// TIA Portal V16 export
// export: Created 2024-04-10T09:00:39.579945Z, ExportSetting WithDefaults, DisplayName Totally Integrated Automation Portal, DisplayVersion V16 Update 6, DisplayName TIA Portal Version Control Interface, DisplayVersion V16 Update 2, DisplayName TIA Portal Openness, DisplayVersion V16 Update 6, DisplayName TIA Portal Test Suite Advanced, DisplayVersion V16, DisplayName SINAMICS Startdrive Advanced, DisplayVersion V16 Update 5, DisplayName SINAMICS Startdrive G130, G150, S120, S150, SINAMICS MV, S210, DisplayVersion V16 Update 5, DisplayName SINAMICS Startdrive G110M, G120, G120C, G120D, G120P, G115D, DisplayVersion V16 Update 5, DisplayName STEP 7 Professional, DisplayVersion V16 Update 6, DisplayName STEP 7 Safety, DisplayVersion V16, DisplayName WinCC Advanced, DisplayVersion V16 Update 6
FUNCTION_BLOCK "RH_OUT_1020MU"   // FB40, LAD
TITLE = Set receiver 865MU1020 outputs / Kuljetinpohja
{ S7_Optimized_Access := 'TRUE' }
AUTHOR : JLA
VERSION : 0.1
// stored: AutoNumber true, IsIECCheckEnabled false, IsRetainMemResEnabled false, MemoryReserve 100, SetENOAutomatically false, UDAEnableTagReadback false
   VAR
      Diag : "RMP_UDT_DIAG";   // Device diagnostics / Laitteen diagnostiikka
      Status : "RMP_UDT_DEV_STATUS";   // Device status information / Laitteen tilatieto
      HMI_Status : "RMP_HMI_DEV_STATUS";   // Device status information for HMI
      IO : Struct   // Device inputs and outputs / Laitteen tulot ja lähdöt
         Input : Struct
            Extended : Bool;   // Receiver extended / Kuljettimen turvakytkin
            Retracted : Bool;   // Receiver retracted / Tulovalokenno
            Rolls_coming : Bool;   // Rolls coming to receiver / Poistovalokenno
            Rolls_received : Bool;   // All rolls received / Rulla viivakoodin lukukohdassa
            Man_extend : Bool;   // Manual, receiver extend
            Man_retract : Bool;   // Manual, receiver retract / Seuraavan kuljettimen tulokenno
            Rolls_on_floor : Bool;   // Edellisen kuljettimen poistokenno / Rolls on floor before stopper
            Lidar_Field1 : Bool;   // Area between stop 1010 and Rm
            Lidar_Field2 : Bool;   // Area after stop 1010
            Lidar_Field3 : Bool;   // Conveyor 2030
            In_11 : Bool;
            In_12 : Bool;
            In_13 : Bool;
            In_14 : Bool;
            In_15 : Bool;
            In_16 : Bool;
            In_17 : Bool;
            In_18 : Bool;
            In_19 : Bool;
            In_20 : Bool;
            In_21 : Bool;
            In_22 : Bool;
            In_23 : Bool;
            In_24 : Bool;
            In_25 : Bool;
            In_26 : Bool;
            In_27 : Bool;
            In_28 : Bool;
            In_29 : Bool;
            In_30 : Bool;
            In_31 : Bool;
            In_32 : Bool;
         END_STRUCT;
         Output : Struct
            Receiver_extend : Bool;   // Receiver extend
            Receiver_retract : Bool;   // Receiver retract
            Out_3 : Bool;
            Out_4 : Bool;
            Out_5 : Bool;
            Out_6 : Bool;
            Out_7 : Bool;
            Out_8 : Bool;
            Out_9 : Bool;
            Out_10 : Bool;
            Out_11 : Bool;
            Out_12 : Bool;
            Out_13 : Bool;
            Out_14 : Bool;
            Out_15 : Bool;
            Out_16 : Bool;
            Out_17 : Bool;
            Out_18 : Bool;
            Out_19 : Bool;
            Out_20 : Bool;
            Out_21 : Bool;
            Out_22 : Bool;
            Out_23 : Bool;
            Out_24 : Bool;
            Out_25 : Bool;
            Out_26 : Bool;
            Out_27 : Bool;
            Out_28 : Bool;
            Out_29 : Bool;
            Out_30 : Bool;
            Out_31 : Bool;
            Out_32 : Bool;
         END_STRUCT;
      END_STRUCT;
      Flags : Struct   // Device auxilary flags / Laitteen apubitit
         Speed_1 : Bool;   // Speed selection 1 / Nopeusvalinta 1
         Speed_2 : Bool;   // Speed selection 2 / Nopeusvalinta 2
         Speed_3 : Bool;   // Speed selection 3 / Nopeusvalinta 3
         Speed_4 : Bool;   // Speed selection 4 / Nopeusvalinta 4
         Data_ok : Bool;   // Roll data present / Rulladata löytyy
         Entry_pec_fault : Bool;   // Entry pec fault bit
         Exit_pec_fault : Bool;   // Exit pec fault bit
         Auto_help : Bool;   // Auto status help bit
         Buffering : Bool;   // Buffering rolls on conveyor
         Separate : Bool;   // Separating rolls at conveyor exit joint
         Separate_p : Bool;   // Separating rolls at conveyor exit joint pulse
         Stopped : Bool;   // Device stopped
         Receiving : Bool;   // Receiving set on conveyor
         Bit_13 : Bool;
         Bit_14 : Bool;
         Bit_15 : Bool;
         Bit_16 : Bool;
         Bit_17 : Bool;
         Bit_18 : Bool;
         Bit_19 : Bool;
         Bit_20 : Bool;
         Bit_21 : Bool;
         Bit_22 : Bool;
         Bit_23 : Bool;
         Bit_24 : Bool;
         Bit_25 : Bool;
         Bit_26 : Bool;
         Bit_27 : Bool;
         Bit_28 : Bool;
         Bit_29 : Bool;
         Bit_30 : Bool;
         Bit_31 : Bool;
         Bit_32 : Bool;
         Bit_33 : Bool;
         Bit_34 : Bool;
         Bit_35 : Bool;
         Bit_36 : Bool;
         Bit_37 : Bool;
         Bit_38 : Bool;
         Bit_39 : Bool;
         Bit_40 : Bool;
         Bit_41 : Bool;
         Bit_42 : Bool;
         Bit_43 : Bool;
         Bit_44 : Bool;
         Bit_45 : Bool;
         Bit_46 : Bool;
         Bit_47 : Bool;
         Bit_48 : Bool;
         Bit_49 : Bool;
         Bit_50 : Bool;
         Bit_51 : Bool;
         Bit_52 : Bool;
         Bit_53 : Bool;
         Bit_54 : Bool;
         Bit_55 : Bool;
         Bit_56 : Bool;
         Bit_57 : Bool;
         Bit_58 : Bool;
         Bit_59 : Bool;
         Bit_60 : Bool;
         Bit_61 : Bool;
         Bit_62 : Bool;
         Bit_63 : Bool;
      END_STRUCT;
      Data : Struct   // Device data / Laitteen data
         Data_int_1 : Int;
         Data_int_2 : Int;
         Data_int_3 : Int;
         Data_int_4 : Int;
         Data_int_5 : Int;
         Data_int_6 : Int;
         Data_int_7 : Int;
         Data_int_8 : Int;
         Data_int_9 : Int;
         Data_int_10 : Int;
         Data_int_11 : Int;
         Data_int_12 : Int;
         Data_int_13 : Int;
         Data_int_14 : Int;
         Data_int_15 : Int;
         Data_int_16 : Int;
         Data_int_17 : Int;
         Data_int_18 : Int;
         Data_int_19 : Int;
         Data_int_20 : Int;
         Data_Dint_1 : DInt;
         Data_Dint_2 : DInt;
         Data_Dint_3 : DInt;
         Data_Dint_4 : DInt;
         Data_Dint_5 : DInt;
         Data_Dint_6 : DInt;
         Data_Dint_7 : DInt;
         Data_Dint_8 : DInt;
         Data_Dint_9 : DInt;
         Data_Dint_10 : DInt;
         Data_Dint_11 : DInt;
         Data_Dint_12 : DInt;
         Data_Dint_13 : DInt;
         Data_Dint_14 : DInt;
         Data_Dint_15 : DInt;
         Data_Dint_16 : DInt;
         Data_from_prev : DWord;   // Data from previous conveyor
         Data_from_next : DWord;   // Data from next conveyor
         Data_next : DWord;   // Conveyor data for next conveyor / Kuljettimen data seuraavalle kuljettimelle
         Data_prev : DWord;   // Conveyor data for previous conveyor / Kuljettimen data edelliselle kuljettimelle
      END_STRUCT;
      Interlock : "RMP_UDT_INTERLOCK";   // Set receiver / Laitelukitukset
      Control : "RMP_UDT_CONTROL";   // Laitteen ohjaus / Device control
      Program_Alarm : Array[1..16] of Program_Alarm;   // Device alarms
      Program_Event : Array[1..8] of Program_Alarm;   // Device events / Laitteen tapahtumat
      Device_name : String[40] := 'Set receiver - 865MU1020';   // Device name
      Fault_1_delay : TON_TIME;
      Event_1_delay : TON_TIME;
      ORG : Struct
         ORG_1 : Bool;   // Data Ready
         ORG_2 : Bool;
         ORG_3 : Bool;
         ORG_4 : Bool;
         ORG_5 : Bool;
         ORG_6 : Bool;
         ORG_7 : Bool;
         ORG_8 : Bool;
      END_STRUCT;
      "865MU1020GL2 Delay" { S7_SetPoint := 'True'} : TON_TIME;
      Extra_valve { S7_SetPoint := 'True'} : TON_TIME;
      Extended_delay { S7_SetPoint := 'True'} : TON_TIME;
      "865MU1020GL1_Delay" { S7_SetPoint := 'True'} : TON_TIME;
      Roll_Detect_Delay { S7_SetPoint := 'True'} : TON_TIME;
      Filter_Lidar_Field1 { S7_SetPoint := 'True'} : TON_TIME;
      Filter_Lidar_Field2 { S7_SetPoint := 'True'} : TON_TIME;
      Filter_Lidar_Field3 { S7_SetPoint := 'True'} : TON_TIME;
      Receiving_delay { S7_SetPoint := 'True'} : TON_TIME;
   END_VAR
   VAR_TEMP
      Temp_R : Real;
      Temp_I : Int;
      Temp_DI : DInt;
      Error : Bool;
      Error_nbr : Int;
   END_VAR
   // // Interlock.Fwd : eteenpäin / to front interlocks
   // // Interlock.Fwd[1] : Conveyor sequence not ready
   // // Interlock.Fwd[2] : Conveyor not empty
   // // Interlock.Fwd[3] : Conveyor running
   // // Interlock.Fwd[4] : Conveyor entry pec
   // // Interlock.Fwd[5] : Conveyor exit pec
   // // Interlock.Fwd[6] : Rapid Door is not closed
   // // Interlock.Rev : taaksepäin / to back interlocks
   // // Interlock.Rev[1] : Rapid door is not closed
   VAR_TEMP   // added for the SCL form of the ladder/FBD networks
      _w1 : Bool;
   END_VAR
BEGIN

REGION Network 1: Control area interface / Ohjausalueen rajapinta
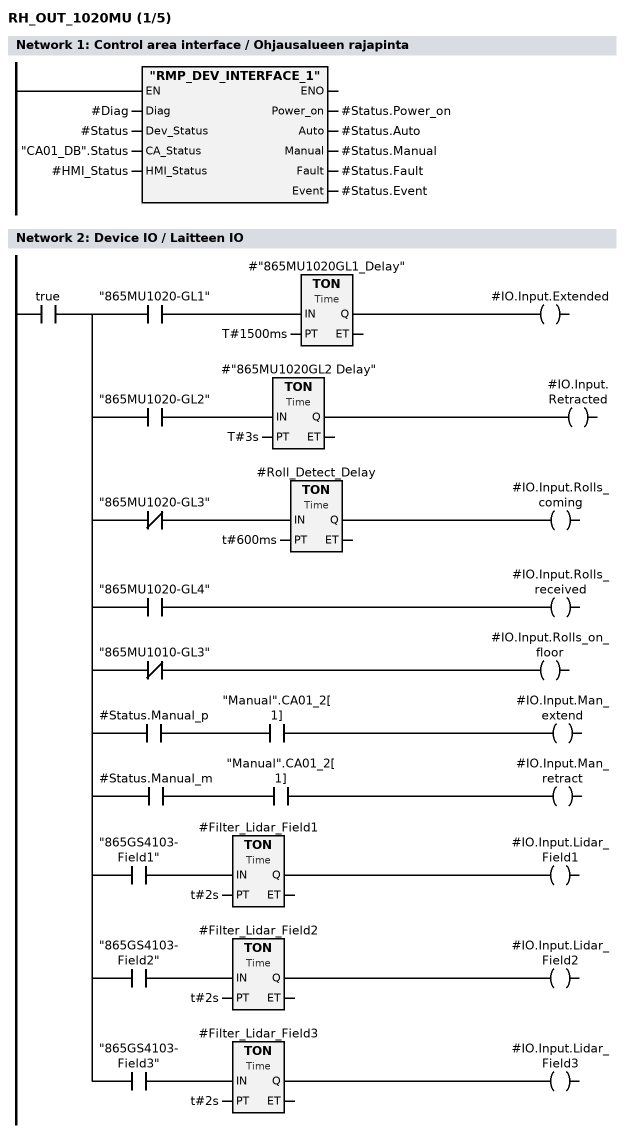
   RUNG wire#powerrail
      "RMP_DEV_INTERFACE_1"(Diag := #Diag, Dev_Status := #Status, CA_Status := "CA01_DB".Status, HMI_Status := #HMI_Status, Power_on => #Status.Power_on, Auto => #Status.Auto, Manual => #Status.Manual, Fault => #Status.Fault, Event => #Status.Event)
   END_RUNG
   // the same network as SCL:
   "RMP_DEV_INTERFACE_1"(Diag := #Diag,
                         Dev_Status := #Status,
                         CA_Status := "CA01_DB".Status,
                         HMI_Status := #HMI_Status,
                         Power_on => #Status.Power_on,
                         Auto => #Status.Auto,
                         Manual => #Status.Manual,
                         Fault => #Status.Fault,
                         Event => #Status.Event);
END_REGION

REGION Network 2: Device IO / Laitteen IO
   RUNG wire#powerrail
      Contact( true )
      wire#w1
      Contact( "865MU1020-GL1" )
      { S7_Templates := "time_type := Time" } #"865MU1020GL1_Delay".TON(pt := T#1500ms, et =>)
      Coil( #IO.Input.Extended )
   END_RUNG
   RUNG wire#w1
      Contact( "865MU1020-GL2" )
      { S7_Templates := "time_type := Time" } #"865MU1020GL2 Delay".TON(pt := T#3s, et =>)
      Coil( #IO.Input.Retracted )
   END_RUNG
   RUNG wire#w1
      I_Contact( "865MU1020-GL3" )
      { S7_Templates := "time_type := Time" } #Roll_Detect_Delay.TON(pt := t#600ms, et =>)
      Coil( #IO.Input.Rolls_coming )
   END_RUNG
   RUNG wire#w1
      Contact( "865MU1020-GL4" )
      Coil( #IO.Input.Rolls_received )
   END_RUNG
   RUNG wire#w1
      I_Contact( "865MU1010-GL3" )
      Coil( #IO.Input.Rolls_on_floor )
   END_RUNG
   RUNG wire#w1
      Contact( #Status.Manual_p )
      Contact( "Manual".CA01_2[1] )
      Coil( #IO.Input.Man_extend )
   END_RUNG
   RUNG wire#w1
      Contact( #Status.Manual_m )
      Contact( "Manual".CA01_2[1] )
      Coil( #IO.Input.Man_retract )
   END_RUNG
   RUNG wire#w1
      Contact( "865GS4103-Field1" )
      { S7_Templates := "time_type := Time" } #Filter_Lidar_Field1.TON(pt := t#2s, et =>)
      Coil( #IO.Input.Lidar_Field1 )
   END_RUNG
   RUNG wire#w1
      Contact( "865GS4103-Field2" )
      { S7_Templates := "time_type := Time" } #Filter_Lidar_Field2.TON(pt := t#2s, et =>)
      Coil( #IO.Input.Lidar_Field2 )
   END_RUNG
   RUNG wire#w1
      Contact( "865GS4103-Field3" )
      { S7_Templates := "time_type := Time" } #Filter_Lidar_Field3.TON(pt := t#2s, et =>)
      Coil( #IO.Input.Lidar_Field3 )
   END_RUNG
   // the same network as SCL:
   #"865MU1020GL1_Delay"(IN := true AND "865MU1020-GL1", PT := T#1500ms);   // TON
   #IO.Input.Extended := #"865MU1020GL1_Delay".Q;
   #"865MU1020GL2 Delay"(IN := true AND "865MU1020-GL2", PT := T#3s);   // TON
   #IO.Input.Retracted := #"865MU1020GL2 Delay".Q;
   #Roll_Detect_Delay(IN := true AND NOT "865MU1020-GL3", PT := t#600ms);   // TON
   #IO.Input.Rolls_coming := #Roll_Detect_Delay.Q;
   #IO.Input.Rolls_received := true AND "865MU1020-GL4";
   #IO.Input.Rolls_on_floor := true AND NOT "865MU1010-GL3";
   #IO.Input.Man_extend := true AND #Status.Manual_p AND "Manual".CA01_2[1];
   #IO.Input.Man_retract := true AND #Status.Manual_m AND "Manual".CA01_2[1];
   #Filter_Lidar_Field1(IN := true AND "865GS4103-Field1", PT := t#2s);   // TON
   #IO.Input.Lidar_Field1 := #Filter_Lidar_Field1.Q;
   #Filter_Lidar_Field2(IN := true AND "865GS4103-Field2", PT := t#2s);   // TON
   #IO.Input.Lidar_Field2 := #Filter_Lidar_Field2.Q;
   #Filter_Lidar_Field3(IN := true AND "865GS4103-Field3", PT := t#2s);   // TON
   #IO.Input.Lidar_Field3 := #Filter_Lidar_Field3.Q;
END_REGION

REGION Network 3: Device sequence
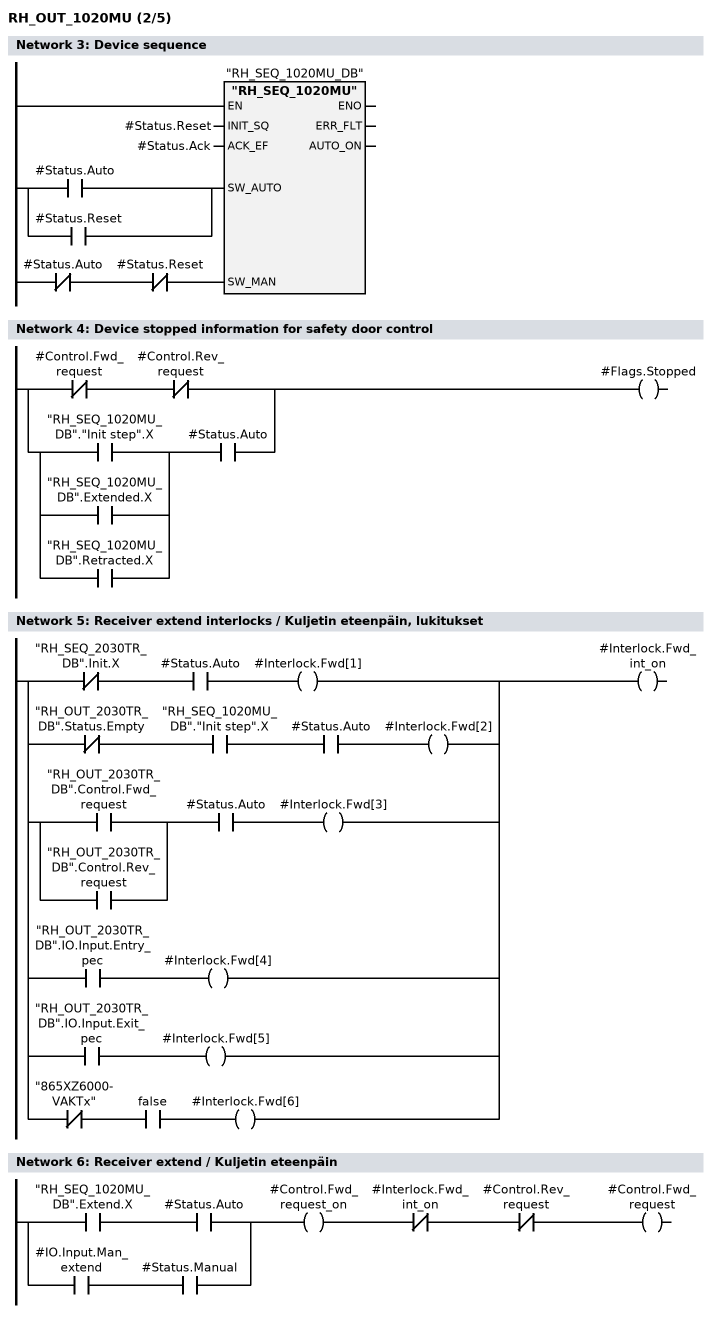
   RUNG wire#powerrail
      "RH_SEQ_1020MU_DB"(SW_AUTO := wire#w1, SW_MAN := wire#w2, INIT_SQ := #Status.Reset, ACK_EF := #Status.Ack, ERR_FLT =>, AUTO_ON =>)
   END_RUNG
   RUNG wire#powerrail
      Contact( #Status.Auto )
   END_RUNG wire#w1
   RUNG wire#powerrail
      Contact( #Status.Reset )
   END_RUNG wire#w1
   RUNG wire#powerrail
      I_Contact( #Status.Auto )
      I_Contact( #Status.Reset )
   END_RUNG wire#w2
   // the same network as SCL:
   "RH_SEQ_1020MU_DB"(INIT_SQ := #Status.Reset,   // "RH_SEQ_1020MU"
                      ACK_EF := #Status.Ack,
                      SW_AUTO := #Status.Auto OR #Status.Reset,
                      SW_MAN := NOT #Status.Auto AND NOT #Status.Reset);
END_REGION

REGION Network 4: Device stopped information for safety door control
   RUNG wire#powerrail
      I_Contact( #Control.Fwd_request )
      I_Contact( #Control.Rev_request )
      wire#w1
      Coil( #Flags.Stopped )
   END_RUNG
   RUNG wire#powerrail
      Contact( "RH_SEQ_1020MU_DB"."Init step".X )
      wire#w2
      Contact( #Status.Auto )
   END_RUNG wire#w1
   RUNG wire#powerrail
      Contact( "RH_SEQ_1020MU_DB".Extended.X )
   END_RUNG wire#w2
   RUNG wire#powerrail
      Contact( "RH_SEQ_1020MU_DB".Retracted.X )
   END_RUNG wire#w2
   // the same network as SCL:
   #Flags.Stopped := (NOT #Control.Fwd_request AND NOT #Control.Rev_request) OR (("RH_SEQ_1020MU_DB"."Init step".X OR "RH_SEQ_1020MU_DB".Extended.X OR "RH_SEQ_1020MU_DB".Retracted.X) AND #Status.Auto);
END_REGION

REGION Network 5: Receiver extend interlocks / Kuljetin eteenpäin, lukitukset
   RUNG wire#powerrail
      I_Contact( "RH_SEQ_2030TR_DB".Init.X )
      Contact( #Status.Auto )
      Coil( #Interlock.Fwd[1] )
      wire#w1
      Coil( #Interlock.Fwd_int_on )
   END_RUNG
   RUNG wire#powerrail
      I_Contact( "RH_OUT_2030TR_DB".Status.Empty )
      Contact( "RH_SEQ_1020MU_DB"."Init step".X )
      Contact( #Status.Auto )
      Coil( #Interlock.Fwd[2] )
   END_RUNG wire#w1
   RUNG wire#powerrail
      Contact( "RH_OUT_2030TR_DB".Control.Fwd_request )
      wire#w2
      Contact( #Status.Auto )
      Coil( #Interlock.Fwd[3] )
   END_RUNG wire#w1
   RUNG wire#powerrail
      Contact( "RH_OUT_2030TR_DB".Control.Rev_request )
   END_RUNG wire#w2
   RUNG wire#powerrail
      Contact( "RH_OUT_2030TR_DB".IO.Input.Entry_pec )
      Coil( #Interlock.Fwd[4] )
   END_RUNG wire#w1
   RUNG wire#powerrail
      Contact( "RH_OUT_2030TR_DB".IO.Input.Exit_pec )
      Coil( #Interlock.Fwd[5] )
   END_RUNG wire#w1
   RUNG wire#powerrail
      I_Contact( "865XZ6000-VAKTx" )
      Contact( false )
      Coil( #Interlock.Fwd[6] )
   END_RUNG wire#w1
   // the same network as SCL:
   #Interlock.Fwd[1] := NOT "RH_SEQ_2030TR_DB".Init.X AND #Status.Auto;
   #Interlock.Fwd[2] := NOT "RH_OUT_2030TR_DB".Status.Empty AND "RH_SEQ_1020MU_DB"."Init step".X AND #Status.Auto;
   #Interlock.Fwd[3] := ("RH_OUT_2030TR_DB".Control.Fwd_request OR "RH_OUT_2030TR_DB".Control.Rev_request) AND #Status.Auto;
   #Interlock.Fwd[4] := "RH_OUT_2030TR_DB".IO.Input.Entry_pec;
   #Interlock.Fwd[5] := "RH_OUT_2030TR_DB".IO.Input.Exit_pec;
   #Interlock.Fwd[6] := NOT "865XZ6000-VAKTx" AND false;
   #Interlock.Fwd_int_on := (NOT "RH_SEQ_2030TR_DB".Init.X AND #Status.Auto) OR (NOT "RH_OUT_2030TR_DB".Status.Empty AND "RH_SEQ_1020MU_DB"."Init step".X AND #Status.Auto) OR (("RH_OUT_2030TR_DB".Control.Fwd_request OR "RH_OUT_2030TR_DB".Control.Rev_request) AND #Status.Auto) OR "RH_OUT_2030TR_DB".IO.Input.Entry_pec OR "RH_OUT_2030TR_DB".IO.Input.Exit_pec OR (NOT "865XZ6000-VAKTx" AND false);
END_REGION

REGION Network 6: Receiver extend / Kuljetin eteenpäin
   RUNG wire#powerrail
      Contact( "RH_SEQ_1020MU_DB".Extend.X )
      Contact( #Status.Auto )
      wire#w1
      Coil( #Control.Fwd_request_on )
      I_Contact( #Interlock.Fwd_int_on )
      I_Contact( #Control.Rev_request )
      Coil( #Control.Fwd_request )
   END_RUNG
   RUNG wire#powerrail
      Contact( #IO.Input.Man_extend )
      Contact( #Status.Manual )
   END_RUNG wire#w1
   // the same network as SCL:
   #Control.Fwd_request_on := ("RH_SEQ_1020MU_DB".Extend.X AND #Status.Auto) OR (#IO.Input.Man_extend AND #Status.Manual);
   #Control.Fwd_request := #Control.Fwd_request_on AND NOT #Interlock.Fwd_int_on AND NOT #Control.Rev_request;
END_REGION

REGION Network 7: Receiver retract interlocks / Kuljetin taaksepäin, lukitukset
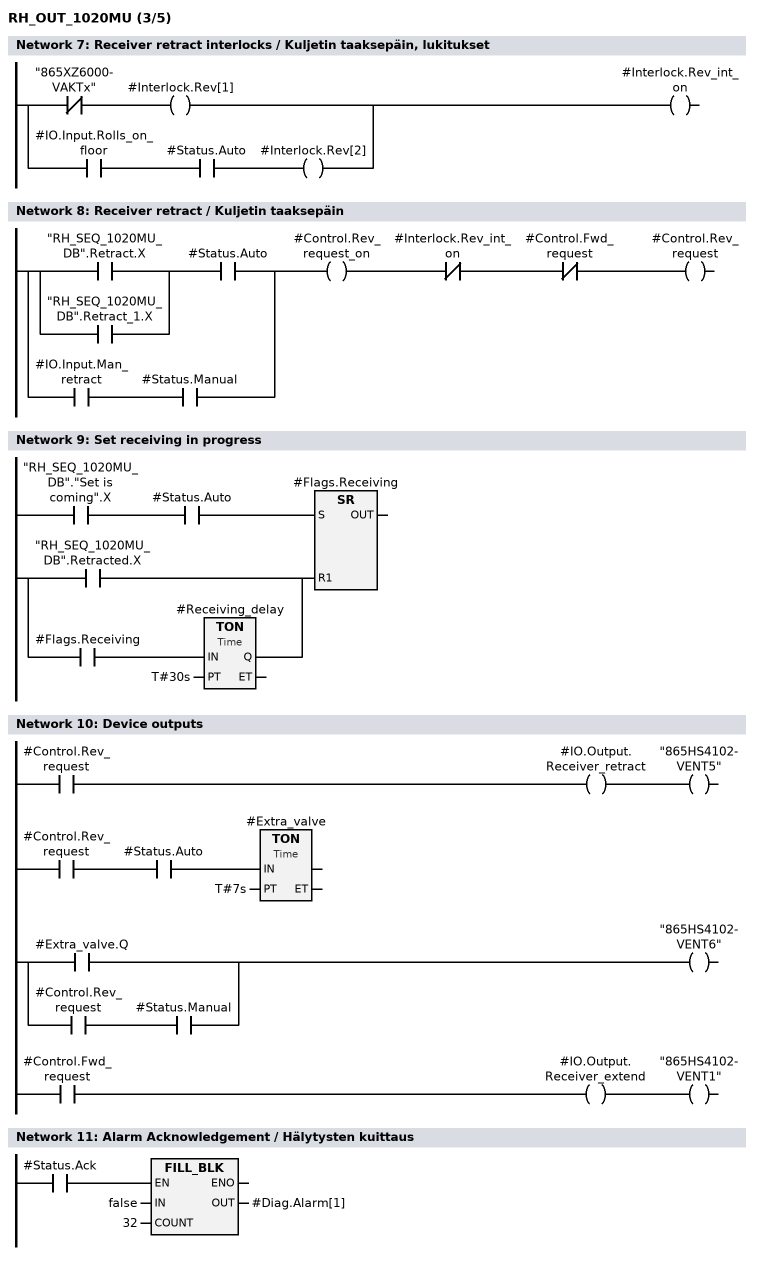
   RUNG wire#powerrail
      I_Contact( "865XZ6000-VAKTx" )
      Coil( #Interlock.Rev[1] )
      wire#w1
      Coil( #Interlock.Rev_int_on )
   END_RUNG
   RUNG wire#powerrail
      Contact( #IO.Input.Rolls_on_floor )
      Contact( #Status.Auto )
      Coil( #Interlock.Rev[2] )
   END_RUNG wire#w1
   // the same network as SCL:
   #Interlock.Rev[1] := NOT "865XZ6000-VAKTx";
   #Interlock.Rev[2] := #IO.Input.Rolls_on_floor AND #Status.Auto;
   #Interlock.Rev_int_on := NOT "865XZ6000-VAKTx" OR (#IO.Input.Rolls_on_floor AND #Status.Auto);
END_REGION

REGION Network 8: Receiver retract / Kuljetin taaksepäin
   RUNG wire#powerrail
      Contact( "RH_SEQ_1020MU_DB".Retract.X )
      wire#w1
      Contact( #Status.Auto )
      wire#w2
      Coil( #Control.Rev_request_on )
      I_Contact( #Interlock.Rev_int_on )
      I_Contact( #Control.Fwd_request )
      Coil( #Control.Rev_request )
   END_RUNG
   RUNG wire#powerrail
      Contact( "RH_SEQ_1020MU_DB".Retract_1.X )
   END_RUNG wire#w1
   RUNG wire#powerrail
      Contact( #IO.Input.Man_retract )
      Contact( #Status.Manual )
   END_RUNG wire#w2
   // the same network as SCL:
   #Control.Rev_request_on := (("RH_SEQ_1020MU_DB".Retract.X OR "RH_SEQ_1020MU_DB".Retract_1.X) AND #Status.Auto) OR (#IO.Input.Man_retract AND #Status.Manual);
   #Control.Rev_request := #Control.Rev_request_on AND NOT #Interlock.Rev_int_on AND NOT #Control.Fwd_request;
END_REGION

REGION Network 9: Set receiving in progress
   RUNG wire#powerrail
      Contact( "RH_SEQ_1020MU_DB"."Set is coming".X )
      Contact( #Status.Auto )
      S_SR(operand := #Flags.Receiving, r1 := wire#w1)
   END_RUNG
   RUNG wire#powerrail
      Contact( "RH_SEQ_1020MU_DB".Retracted.X )
   END_RUNG wire#w1
   RUNG wire#powerrail
      Contact( #Flags.Receiving )
      { S7_Templates := "time_type := Time" } #Receiving_delay.TON(pt := T#30s, et =>)
   END_RUNG wire#w1
   // the same network as SCL:
   #Receiving_delay(IN := #Flags.Receiving, PT := T#30s);   // TON
   IF "RH_SEQ_1020MU_DB"."Set is coming".X AND #Status.Auto THEN
       #Flags.Receiving := TRUE;   // SR flip-flop
   END_IF;
   IF "RH_SEQ_1020MU_DB".Retracted.X OR #Receiving_delay.Q THEN #Flags.Receiving := FALSE; END_IF;
END_REGION

REGION Network 10: Device outputs
   RUNG wire#powerrail
      Contact( #Control.Rev_request )
      Coil( #IO.Output.Receiver_retract )
      Coil( "865HS4102-VENT5" )
   END_RUNG
   RUNG wire#powerrail
      Contact( #Control.Rev_request )
      Contact( #Status.Auto )
      { S7_Templates := "time_type := Time" } #Extra_valve.TON(pt := T#7s, et =>)
   END_RUNG
   RUNG wire#powerrail
      Contact( #Extra_valve.Q )
      wire#w1
      Coil( "865HS4102-VENT6" )
   END_RUNG
   RUNG wire#powerrail
      Contact( #Control.Rev_request )
      Contact( #Status.Manual )
   END_RUNG wire#w1
   RUNG wire#powerrail
      Contact( #Control.Fwd_request )
      Coil( #IO.Output.Receiver_extend )
      Coil( "865HS4102-VENT1" )
   END_RUNG
   // the same network as SCL:
   #IO.Output.Receiver_retract := #Control.Rev_request;
   "865HS4102-VENT5" := #Control.Rev_request;
   #Extra_valve(IN := #Control.Rev_request AND #Status.Auto, PT := T#7s);   // TON
   "865HS4102-VENT6" := #Extra_valve.Q OR (#Control.Rev_request AND #Status.Manual);
   #IO.Output.Receiver_extend := #Control.Fwd_request;
   "865HS4102-VENT1" := #Control.Fwd_request;
END_REGION

REGION Network 11: Alarm Acknowledgement / Hälytysten kuittaus
   RUNG wire#powerrail
      Contact( #Status.Ack )
      FillBlockI(in := false, count := 32, out => #Diag.Alarm[1])
   END_RUNG
   // the same network as SCL:
   IF #Status.Ack THEN FILL_BLK(IN := false, COUNT := 32, OUT => #Diag.Alarm[1]); END_IF;
END_REGION

REGION Network 12: Alarm 1: Set receiver limit switch fault / Taajuusmuuttajan vika
   // Taajuusmuuttajan vika
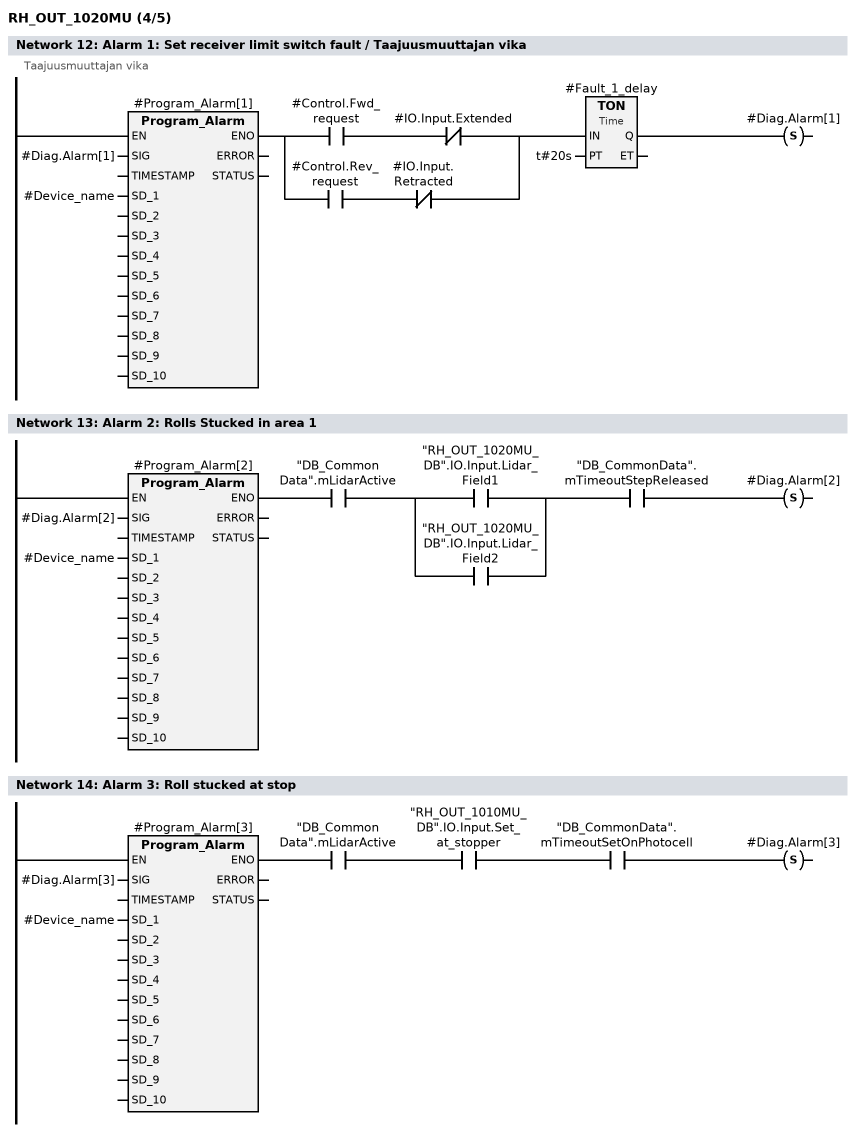
   RUNG wire#powerrail
      #Program_Alarm[1].Program_Alarm(SIG := #Diag.Alarm[1], TIMESTAMP :=, SD_1 := #Device_name, SD_2 :=, SD_3 :=, SD_4 :=, SD_5 :=, SD_6 :=, SD_7 :=, SD_8 :=, SD_9 :=, SD_10 :=, Error =>, Status =>)
      wire#w1
      Contact( #Control.Fwd_request )
      I_Contact( #IO.Input.Extended )
      wire#w2
      { S7_Templates := "time_type := Time" } #Fault_1_delay.TON(pt := t#20s, et =>)
      S_Coil( #Diag.Alarm[1] )
   END_RUNG
   RUNG wire#w1
      Contact( #Control.Rev_request )
      I_Contact( #IO.Input.Retracted )
   END_RUNG wire#w2
   // the same network as SCL:
   #Program_Alarm[1](SIG := #Diag.Alarm[1], SD_1 := #Device_name, ENO => #_w1);   // Program_Alarm
   #Fault_1_delay(IN := #_w1 AND ((#Control.Fwd_request AND NOT #IO.Input.Extended) OR (#Control.Rev_request AND NOT #IO.Input.Retracted)),   // TON
                  PT := t#20s);
   IF #Fault_1_delay.Q THEN #Diag.Alarm[1] := TRUE; END_IF;
END_REGION

REGION Network 13: Alarm 2: Rolls Stucked in area 1
   RUNG wire#powerrail
      #Program_Alarm[2].Program_Alarm(SIG := #Diag.Alarm[2], TIMESTAMP :=, SD_1 := #Device_name, SD_2 :=, SD_3 :=, SD_4 :=, SD_5 :=, SD_6 :=, SD_7 :=, SD_8 :=, SD_9 :=, SD_10 :=, Error =>, Status =>)
      Contact( "DB_CommonData".mLidarActive )
      wire#w1
      Contact( "RH_OUT_1020MU_DB".IO.Input.Lidar_Field1 )
      wire#w2
      Contact( "DB_CommonData".mTimeoutStepReleased )
      S_Coil( #Diag.Alarm[2] )
   END_RUNG
   RUNG wire#w1
      Contact( "RH_OUT_1020MU_DB".IO.Input.Lidar_Field2 )
   END_RUNG wire#w2
   // the same network as SCL:
   #Program_Alarm[2](SIG := #Diag.Alarm[2], SD_1 := #Device_name, ENO => #_w1);   // Program_Alarm
   IF #_w1 AND "DB_CommonData".mLidarActive AND ("RH_OUT_1020MU_DB".IO.Input.Lidar_Field1 OR "RH_OUT_1020MU_DB".IO.Input.Lidar_Field2) AND "DB_CommonData".mTimeoutStepReleased THEN
       #Diag.Alarm[2] := TRUE;
   END_IF;
END_REGION

REGION Network 14: Alarm 3: Roll stucked at stop
   RUNG wire#powerrail
      #Program_Alarm[3].Program_Alarm(SIG := #Diag.Alarm[3], TIMESTAMP :=, SD_1 := #Device_name, SD_2 :=, SD_3 :=, SD_4 :=, SD_5 :=, SD_6 :=, SD_7 :=, SD_8 :=, SD_9 :=, SD_10 :=, Error =>, Status =>)
      Contact( "DB_CommonData".mLidarActive )
      Contact( "RH_OUT_1010MU_DB".IO.Input.Set_at_stopper )
      Contact( "DB_CommonData".mTimeoutSetOnPhotocell )
      S_Coil( #Diag.Alarm[3] )
   END_RUNG
   // the same network as SCL:
   #Program_Alarm[3](SIG := #Diag.Alarm[3], SD_1 := #Device_name, ENO => #_w1);   // Program_Alarm
   IF #_w1 AND "DB_CommonData".mLidarActive AND "RH_OUT_1010MU_DB".IO.Input.Set_at_stopper AND "DB_CommonData".mTimeoutSetOnPhotocell THEN
       #Diag.Alarm[3] := TRUE;
   END_IF;
END_REGION

REGION Network 15: Event 1:Device interlock on / Laitteen lukitus päällä
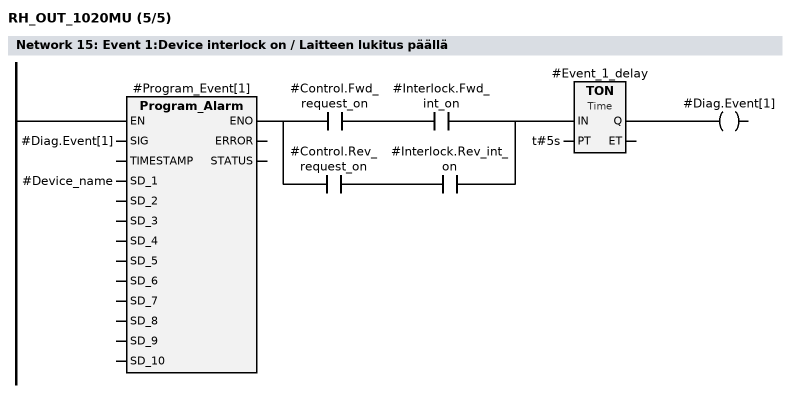
   RUNG wire#powerrail
      #Program_Event[1].Program_Alarm(SIG := #Diag.Event[1], TIMESTAMP :=, SD_1 := #Device_name, SD_2 :=, SD_3 :=, SD_4 :=, SD_5 :=, SD_6 :=, SD_7 :=, SD_8 :=, SD_9 :=, SD_10 :=, Error =>, Status =>)
      wire#w1
      Contact( #Control.Fwd_request_on )
      Contact( #Interlock.Fwd_int_on )
      wire#w2
      { S7_Templates := "time_type := Time" } #Event_1_delay.TON(pt := t#5s, et =>)
      Coil( #Diag.Event[1] )
   END_RUNG
   RUNG wire#w1
      Contact( #Control.Rev_request_on )
      Contact( #Interlock.Rev_int_on )
   END_RUNG wire#w2
   // the same network as SCL:
   #Program_Event[1](SIG := #Diag.Event[1], SD_1 := #Device_name, ENO => #_w1);   // Program_Alarm
   #Event_1_delay(IN := #_w1 AND ((#Control.Fwd_request_on AND #Interlock.Fwd_int_on) OR (#Control.Rev_request_on AND #Interlock.Rev_int_on)),   // TON
                  PT := t#5s);
   #Diag.Event[1] := #Event_1_delay.Q;
END_REGION
END_FUNCTION_BLOCK
